Fanuc KAREL source: ko00050.KL

-- PROVISIONAL review KL for V1013-1; original PC SHA256 868036d132ae2f62fae20cc3a10313b8ff62935b31478bf5203a30a71a7a9978
-- Incomplete behavior may be omitted. Consult companion uncertainty JSON. Do not deploy.
PROGRAM KO00050
%NOLOCKGROUP
BEGIN
  -- UNRESOLVED_PC offsets 5-12; opcodes 9D,23
  -- UNRESOLVED_PC offsets 17-66; opcodes 27,27,49,7E,AD,22,1C,22,31,7E,4A
  -- UNRESOLVED_PC offsets 71-75; opcodes 7F
END KO00050
